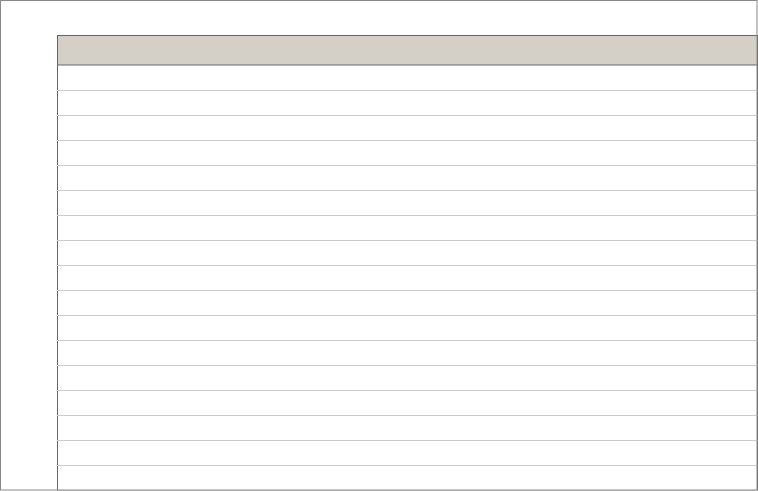
VISUALIZATION alarmHist  // 758x491
    Table (57,35 701x456), data array: toHMI.aHist
        p3854506369: toHMI.aHist[INDEX].sDate
        p1892666644: toHMI.aHist[INDEX].sTime
        p338671338: toHMI.aHist[INDEX].sMessage
END_VISUALIZATION

(* stored: Version 1.1.0.1, ProductVersion 3.1.4024.11
   Visu alarmHist: Id {bc3245b3-b89d-4103-bdfe-1016d41c083e} *)
